FUNCTION_BLOCK Equipo_Valvula_5_2_biestable
VAR_INPUT
	PE				:BOOL; //Parada de emergência
	Modo_Automatico	:BOOL;	//Modo automático
	Cmd_Auto_Pos1	:BOOL;	//Comando para a posição 1
	Cmd_Auto_Pos2	:BOOL;	//Comando para a posição 2
	Valv_Pos1		:BOOL;	//Válvula na posição 1
	Valv_Pos2		:BOOL;	//Válvula na posição 2
	T_Discrepancia	:TIME;	//Tempo para falha na abertura
END_VAR
VAR_OUTPUT
	Activa_Pos1			:BOOL;	//Aciona a saída para a posição 1
	Activa_Pos2			:BOOL;	//Aciona a saída para a posição 2
	Estado				:INT;	//Estado da válvula
	Alr_Discrepancia	:BOOL;	//Em alarme
END_VAR
VAR_IN_OUT
	Cmd_Man_Pos1		:BOOL;	//Comando manual para a posição 1
	Cmd_Man_Pos2		:BOOL;	//Comando manual para a posição 2
	Alarma				:BOOL;	//Em alarme
	Reset_Alarma		:BOOL;	//Reset alarme
END_VAR
VAR_STAT
	FP_Reset			:R_TRIG;	//Borda para reset
	FN_Parada_Auto		:F_TRIG;	//Borda para parada em automático
	FP_Marcha_Auto		:R_TRIG;	//Borda para partir em aitomático
	Cmd_Auto_interno	:BOOL;		//Borda para comando manual
END_VAR

VAR PERSISTENT
	Reset_Eventos		:BOOL;	//Reset contagem de acionamentos
	Timer_Discrepancia		:TON;	//Timer para falha de abertura
	TON_TempoAcionamento	:TON;	//Timer para contar o tempo de acionamento
	R_TRIG_Acionamento		:R_TRIG;	//Borda para tempo de acionamento
	TempoAcionamento		:DINT;	//Tempo de acionamento
	Eventos_Parciales	:DINT;	//Contagem de acionamentos
	Eventos_Totales		:DINT;	//Contagem de eventos totais
END_VAR
VAR // added by the converter: edge detectors and wires of the graphical bodies
    _w1, _w2, _w3, _w4, _w5, _w6, _w7 : BOOL;
    _rt1, _rt2 : R_TRIG;
END_VAR

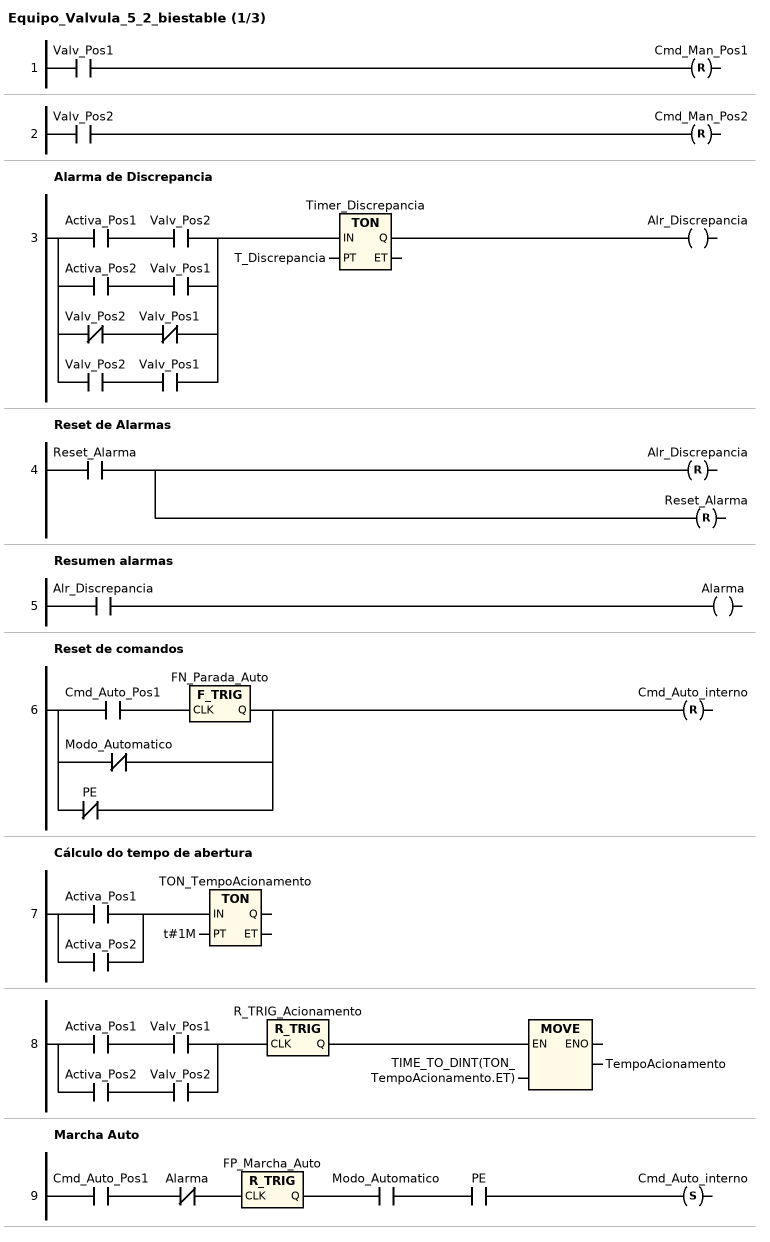
// NETWORK 1
Cmd_Man_Pos1 R= Valv_Pos1;

// NETWORK 2
Cmd_Man_Pos2 R= Valv_Pos2;

// NETWORK 3: Alarma de Discrepancia
Timer_Discrepancia(IN := Activa_Pos1 AND Valv_Pos2 OR Activa_Pos2 AND Valv_Pos1 OR NOT Valv_Pos2 AND NOT Valv_Pos1 OR Valv_Pos2 AND Valv_Pos1, PT := T_Discrepancia); // TON
Alr_Discrepancia := Timer_Discrepancia.Q;

// NETWORK 4: Reset de Alarmas
Alr_Discrepancia R= Reset_Alarma;
Reset_Alarma R= Reset_Alarma;

// NETWORK 5: Resumen alarmas
Alarma := Alr_Discrepancia;

// NETWORK 6: Reset de comandos
FN_Parada_Auto(CLK := Cmd_Auto_Pos1); // F_TRIG
Cmd_Auto_interno R= FN_Parada_Auto.Q OR NOT Modo_Automatico OR NOT PE;

// NETWORK 7: Cálculo do tempo de abertura
TON_TempoAcionamento(IN := Activa_Pos1 OR Activa_Pos2, PT := t#1M); // TON

// NETWORK 8
R_TRIG_Acionamento(CLK := Activa_Pos1 AND Valv_Pos1 OR Activa_Pos2 AND Valv_Pos2); // R_TRIG
IF R_TRIG_Acionamento.Q THEN TempoAcionamento := TIME_TO_DINT(TON_TempoAcionamento.ET); END_IF

// NETWORK 9: Marcha Auto
FP_Marcha_Auto(CLK := Cmd_Auto_Pos1 AND NOT Alarma); // R_TRIG
Cmd_Auto_interno S= FP_Marcha_Auto.Q AND Modo_Automatico AND PE;

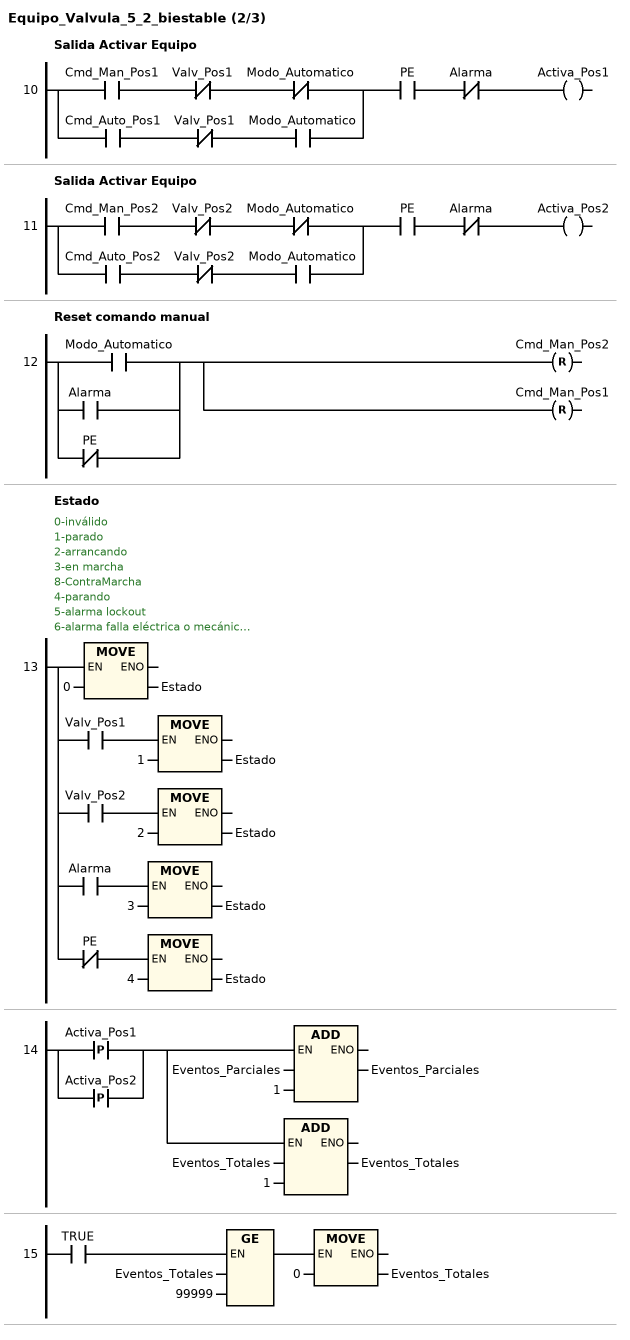
// NETWORK 10: Salida Activar Equipo
Activa_Pos1 := (Cmd_Man_Pos1 AND NOT Valv_Pos1 AND NOT Modo_Automatico OR Cmd_Auto_Pos1 AND NOT Valv_Pos1 AND Modo_Automatico) AND PE AND NOT Alarma;

// NETWORK 11: Salida Activar Equipo
Activa_Pos2 := (Cmd_Man_Pos2 AND NOT Valv_Pos2 AND NOT Modo_Automatico OR Cmd_Auto_Pos2 AND NOT Valv_Pos2 AND Modo_Automatico) AND PE AND NOT Alarma;

// NETWORK 12: Reset comando manual
_w1 := Modo_Automatico OR Alarma OR NOT PE;
Cmd_Man_Pos2 R= _w1;
Cmd_Man_Pos1 R= _w1;

// NETWORK 13: Estado
// 0-inválido
// 1-parado
// 2-arrancando
// 3-en marcha
// 8-ContraMarcha
// 4-parando
// 5-alarma lockout
// 6-alarma falla eléctrica o mecánica
// 7-alarma pulsador emergencia
Estado := 0;
_w2 := Valv_Pos1;
IF _w2 THEN Estado := 1; END_IF
_w3 := Valv_Pos2;
IF _w3 THEN Estado := 2; END_IF
_w4 := Alarma;
IF _w4 THEN Estado := 3; END_IF
_w5 := NOT PE;
IF _w5 THEN Estado := 4; END_IF

// NETWORK 14
_rt1(CLK := Activa_Pos1);
_rt2(CLK := Activa_Pos2);
_w6 := _rt1.Q OR _rt2.Q;
IF _w6 THEN Eventos_Parciales := Eventos_Parciales + 1; END_IF
IF _w6 THEN Eventos_Totales := Eventos_Totales + 1; END_IF

// NETWORK 15
IF Eventos_Totales >= 99999 THEN Eventos_Totales := 0; END_IF

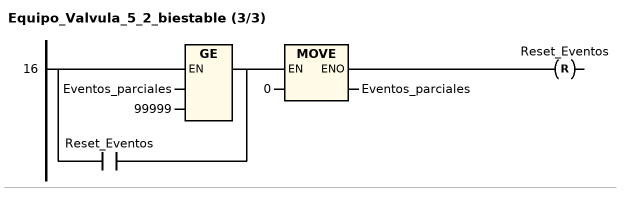
// NETWORK 16
_w7 := Reset_Eventos;
IF NOT _w7 THEN
    _w7 := Eventos_parciales >= 99999;
END_IF
IF _w7 THEN Eventos_parciales := 0; END_IF
Reset_Eventos R= _w7;

END_FUNCTION_BLOCK

(* stored: Version 1.1.0.1, ProductVersion 3.1.4024.14
   POU Equipo_Valvula_5_2_biestable: Id {1946130b-9ea4-49de-8586-e66e0d68a1ad}, SpecialFunc None *)
